// TIA Portal V20 export
TYPE "typeCmControlNodeInterlock"
// stored: Namespace Unit1.Em6
   STRUCT
      hotPressLeftServoPress : "LER_typeServoPressInterlock";
      hotpressLeftStageLiftFront : "LER_typeTwoWayActuatorInterlock";
      hotpressLeftStageLiftRear : "LER_typeTwoWayActuatorInterlock";
      hotpressLeftStageLiftAll : "LER_typeTwoWayActuatorInterlock";
   END_STRUCT;
END_TYPE
